FUNCTION_BLOCK TWOCONRINGTOKEN (* Composite Function Block Type *)
  (* Standard: 61499-2 *)
  (* Version 0.2, 2003-12-05, JHC, Rockwell Automation, Renamed from NEWCOMPFB. *)
  (* Version 0.1, 2002-01-08, JHC, Rockwell Automation, Added DLY FB as example. *)
  (* Version 0.0, 2000-05-27, JHC, Rockwell Automation *)
  (* Compiler header: package fb.rt.cs725; *)
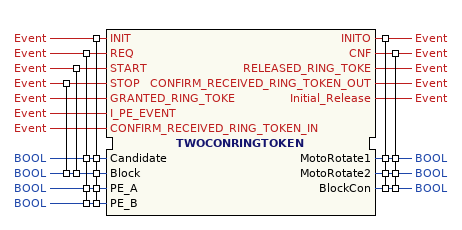
  EVENT_INPUT
    INIT WITH Candidate, Block, PE_A, PE_B; (* Initialization Request *)
    REQ WITH Candidate, PE_A, PE_B; (* Normal Execution Request *)
    START WITH Block;
    STOP WITH Block;
    GRANTED_RING_TOKE;
    I_PE_EVENT;
    CONFIRM_RECEIVED_RING_TOKEN_IN;
  END_EVENT
  EVENT_OUTPUT
    INITO WITH MotoRotate1, MotoRotate2, BlockCon; (* Initialization Confirm *)
    CNF WITH MotoRotate1, MotoRotate2, BlockCon; (* Execution Confirmation *)
    RELEASED_RING_TOKE;
    CONFIRM_RECEIVED_RING_TOKEN_OUT;
    Initial_Release;
  END_EVENT
  VAR_INPUT
    Candidate : BOOL;
    Block : BOOL;
    PE_A : BOOL;
    PE_B : BOOL;
  END_VAR
  VAR_OUTPUT
    MotoRotate1 : BOOL;
    MotoRotate2 : BOOL;
    BlockCon : BOOL;
  END_VAR
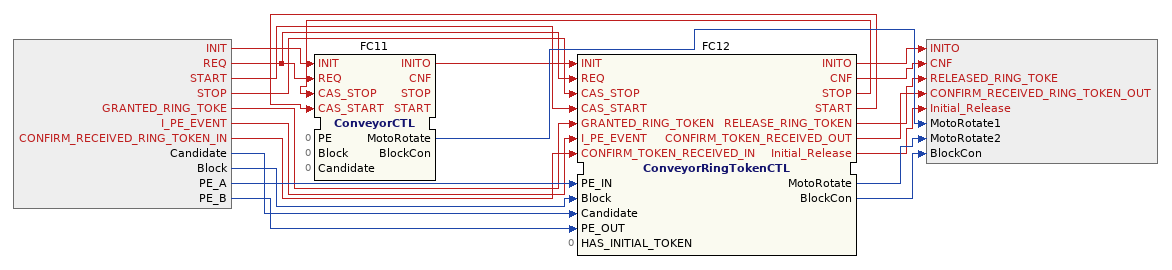
  FBS
    FC11 : ConveyorCTL(Candidate := 0, Block := 0, PE := 0);
    FC12 : ConveyorRingTokenCTL(HAS_INITIAL_TOKEN := 0);
  END_FBS
  EVENT_CONNECTIONS
    INIT TO FC11.INIT;
    REQ TO FC11.REQ;
    FC12.INITO TO INITO;
    FC12.CNF TO CNF;
    REQ TO FC12.REQ;
    STOP TO FC12.CAS_STOP;
    START TO FC12.CAS_START;
    FC12.STOP TO FC11.CAS_STOP;
    FC12.START TO FC11.CAS_START;
    FC11.INITO TO FC12.INIT;
    GRANTED_RING_TOKE TO FC12.GRANTED_RING_TOKEN;
    FC12.RELEASE_RING_TOKEN TO RELEASED_RING_TOKE;
    I_PE_EVENT TO FC12.I_PE_EVENT;
    CONFIRM_RECEIVED_RING_TOKEN_IN TO FC12.CONFIRM_TOKEN_RECEIVED_IN;
    FC12.CONFIRM_TOKEN_RECEIVED_OUT TO CONFIRM_RECEIVED_RING_TOKEN_OUT;
    FC12.Initial_Release TO Initial_Release;
  END_CONNECTIONS
  DATA_CONNECTIONS
    Block TO FC12.Block;
    Candidate TO FC12.Candidate;
    FC12.BlockCon TO BlockCon;
    FC11.MotoRotate TO MotoRotate1;
    FC12.MotoRotate TO MotoRotate2;
    PE_A TO FC12.PE_IN;
    PE_B TO FC12.PE_OUT;
  END_CONNECTIONS
END_FUNCTION_BLOCK
